// TIA Portal V18 export
// export: Created 2025-12-01T17:50:26.9274774Z, ExportSetting None, DisplayName Totally Integrated Automation Portal, DisplayVersion V18 Update 5, DisplayName TIA Portal Openness, DisplayVersion V18 Update 5, DisplayName TIA Portal Teamcenter Gateway, DisplayVersion V18, DisplayName TIA Portal Version Control Interface, DisplayVersion V18, DisplayName STEP 7 Professional, DisplayVersion V18 Update 5, DisplayName STEP 7 Safety, DisplayVersion V18, DisplayName WinCC Professional, DisplayVersion V18 Update 5
FUNCTION_BLOCK "SystemMode"   // FB3000, LAD
TITLE = SystemMode_FB
{ S7_Optimized_Access := 'TRUE' }
AUTHOR : STD
FAMILY : RCS
VERSION : 2.0
// stored: AutoNumber false, MemoryReserve 100, SetENOAutomatically false
   VAR_INPUT
      iPLCRestarted : Bool;
      iEstopAllOK { ExternalAccessible := 'False'; ExternalVisible := 'False'; ExternalWritable := 'False'} : Bool;   // 急停按钮
      iResetFault { ExternalAccessible := 'False'; ExternalVisible := 'False'; ExternalWritable := 'False'} : Bool;   // 故障复位按钮
      iModeSelectType { ExternalAccessible := 'False'; ExternalVisible := 'False'; ExternalWritable := 'False'} : Bool;   // 0=key switch / 1= HMI button
      iManual { ExternalAccessible := 'False'; ExternalVisible := 'False'; ExternalWritable := 'False'} : Bool;   // Key switch signal,1=Manual / Key switch signal,1=Manual Mode
      iAuto { ExternalAccessible := 'False'; ExternalVisible := 'False'; ExternalWritable := 'False'} : Bool;   // Key switch signal,1=Auto / Key switch signal,1=Auto Mode
      iStep { ExternalAccessible := 'False'; ExternalVisible := 'False'; ExternalWritable := 'False'} : Bool;   // Step mode / Auto Step Mode
      iOneCycle : Bool;   // OneCycle / Auto One Cycle Mode
      iHMIModeSelect { ExternalAccessible := 'False'; ExternalVisible := 'False'; ExternalWritable := 'False'} : Int;   // HMI button signal,1=Manual / 2=Auto/3=OneCycle/4=Step / HMI button signal,1=Manual / 2=Auto / 3=Step / 4=OneCyc
      iControlOnMonitor { ExternalAccessible := 'False'; ExternalVisible := 'False'; ExternalWritable := 'False'} : Bool;   // 安全继电器ControlOn监控
      iSafetyDoor { ExternalAccessible := 'False'; ExternalVisible := 'False'; ExternalWritable := 'False'} : Bool;
      iLightCurtain { ExternalAccessible := 'False'; ExternalVisible := 'False'; ExternalWritable := 'False'} : Bool;
      iSafetyByPass : Bool;
      iMainPressureSwitch { ExternalAccessible := 'False'; ExternalVisible := 'False'; ExternalWritable := 'False'} : Bool;   // 主气源开关监控
      iFixtureOK { ExternalAccessible := 'False'; ExternalVisible := 'False'; ExternalWritable := 'False'} : Bool;   // fixture ok
      iChangeOverOK { ExternalAccessible := 'False'; ExternalVisible := 'False'; ExternalWritable := 'False'} : Bool;   // changer over is ok
      iInitializationOK { ExternalAccessible := 'False'; ExternalVisible := 'False'; ExternalWritable := 'False'} : Bool;   // initialization is ok
      iAllDeviceOK { ExternalAccessible := 'False'; ExternalVisible := 'False'; ExternalWritable := 'False'} : Bool;   // all device is ready
      iAlarmOn : Bool;   // 设备故障
      iFlowRun : Bool;   // 设备运行
   END_VAR
   VAR_OUTPUT
      oReset { ExternalAccessible := 'False'; ExternalVisible := 'False'; ExternalWritable := 'False'} : Bool;   // 系统复位信号
      oEStopOK { ExternalAccessible := 'False'; ExternalVisible := 'False'; ExternalWritable := 'False'} : Bool;   // 系统急停控制信号
      oManualMode { ExternalAccessible := 'False'; ExternalVisible := 'False'; ExternalWritable := 'False'} : Bool;   // 手动模式信号
      oAutoMode { ExternalAccessible := 'False'; ExternalVisible := 'False'; ExternalWritable := 'False'} : Bool;   // 自动模式信号
      oOneCycleMode : Bool;   // 单次循环
      oStepMode { ExternalAccessible := 'False'; ExternalVisible := 'False'; ExternalWritable := 'False'} : Bool;
      oRun { ExternalAccessible := 'False'; ExternalVisible := 'False'; ExternalWritable := 'False'} : Bool;   // 系统运行就绪信号 / Control On and all Safety function OK
      "oEnable alarm" : Bool;
      oControlON { ExternalAccessible := 'False'; ExternalVisible := 'False'; ExternalWritable := 'False'} : Bool;   // PowerON
      oMainPressureOK { ExternalAccessible := 'False'; ExternalVisible := 'False'; ExternalWritable := 'False'} : Bool;   // air pressure
      oSafetyDoorOK { ExternalAccessible := 'False'; ExternalVisible := 'False'; ExternalWritable := 'False'} : Bool;   // 安全门关闭
      oLightCurtainOK { ExternalAccessible := 'False'; ExternalVisible := 'False'; ExternalWritable := 'False'} : Bool;   // 光栅
      oReady : Bool;   // 用于流程控制 / In AutoMode and all condition ok, machine can auto running
      oMode { ExternalAccessible := 'False'; ExternalVisible := 'False'; ExternalWritable := 'False'} : Int;   // 0NA,1Manual, 2Auto, 3Step, 4OneCycle, 5Runn, 6Error
      oStatus : Int;   // 0NotReady, 1Ready, 2AutoRunning, 3EStop, 4Alarm
   END_VAR
   VAR
      sRunT { S7_SetPoint := 'True'} : TON_TIME;
      sPressureTOF { S7_SetPoint := 'True'} : TOF_TIME;
      sChangeOverTOF { S7_SetPoint := 'True'} : TOF_TIME;
      sChangeOverOK { S7_SetPoint := 'True'} : Bool;
   END_VAR
   VAR_TEMP
      tAlwaysOn : Bool;
   END_VAR
   VAR_TEMP   // added for the SCL form of the ladder/FBD networks
      _w1 : Bool;
      _w2 : Bool;
      _w3 : Bool;
   END_VAR
BEGIN

REGION Network 1: AlwaysOn
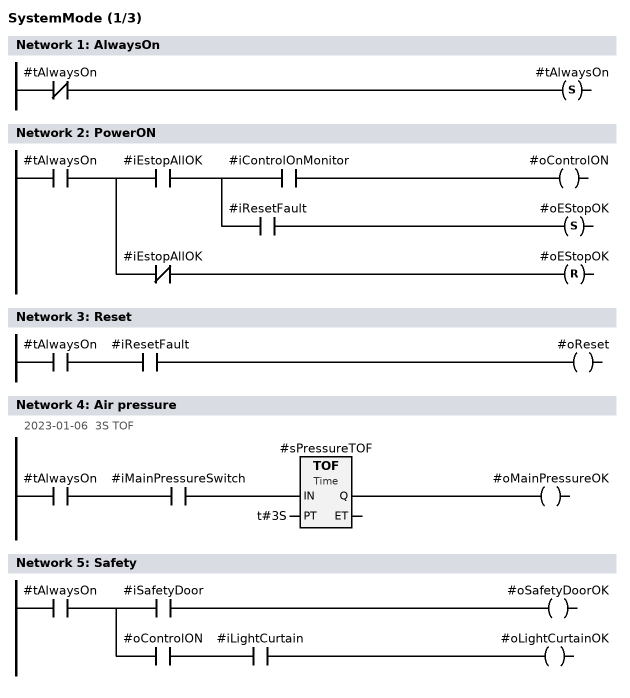
   RUNG wire#powerrail
      I_Contact( #tAlwaysOn )
      S_Coil( #tAlwaysOn )
   END_RUNG
   // the same network as SCL:
   IF NOT #tAlwaysOn THEN #tAlwaysOn := TRUE; END_IF;
END_REGION

REGION Network 2: PowerON
   RUNG wire#powerrail
      Contact( #tAlwaysOn )
      wire#w1
      Contact( #iEstopAllOK )
      wire#w2
      Contact( #iControlOnMonitor )
      Coil( #oControlON )
   END_RUNG
   RUNG wire#w2
      Contact( #iResetFault )
      S_Coil( #oEStopOK )
   END_RUNG
   RUNG wire#w1
      I_Contact( #iEstopAllOK )
      R_Coil( #oEStopOK )
   END_RUNG
   // the same network as SCL:
   #_w1 := #tAlwaysOn AND #iEstopAllOK;
   #oControlON := #_w1 AND #iControlOnMonitor;
   IF #_w1 AND #iResetFault THEN #oEStopOK := TRUE; END_IF;
   IF #tAlwaysOn AND NOT #iEstopAllOK THEN #oEStopOK := FALSE; END_IF;
END_REGION

REGION Network 3: Reset
   RUNG wire#powerrail
      Contact( #tAlwaysOn )
      Contact( #iResetFault )
      Coil( #oReset )
   END_RUNG
   // the same network as SCL:
   #oReset := #tAlwaysOn AND #iResetFault;
END_REGION

REGION Network 4: Air pressure
   // 2023-01-06  3S TOF
   RUNG wire#powerrail
      Contact( #tAlwaysOn )
      Contact( #iMainPressureSwitch )
      { S7_Templates := "time_type := Time" } #sPressureTOF.TOF(pt := t#3S, et =>)
      Coil( #oMainPressureOK )
   END_RUNG
   // the same network as SCL:
   #sPressureTOF(IN := #tAlwaysOn AND #iMainPressureSwitch, PT := t#3S);   // TOF
   #oMainPressureOK := #sPressureTOF.Q;
END_REGION

REGION Network 5: Safety
   RUNG wire#powerrail
      Contact( #tAlwaysOn )
      wire#w1
      Contact( #iSafetyDoor )
      Coil( #oSafetyDoorOK )
   END_RUNG
   RUNG wire#w1
      Contact( #oControlON )
      Contact( #iLightCurtain )
      Coil( #oLightCurtainOK )
   END_RUNG
   // the same network as SCL:
   #oSafetyDoorOK := #tAlwaysOn AND #iSafetyDoor;
   #oLightCurtainOK := #tAlwaysOn AND #oControlON AND #iLightCurtain;
END_REGION

REGION Network 6: Mode
   // 0NA,1Manual, 2Auto, 3Step, 4OneCycle, 5Runn, 6Error
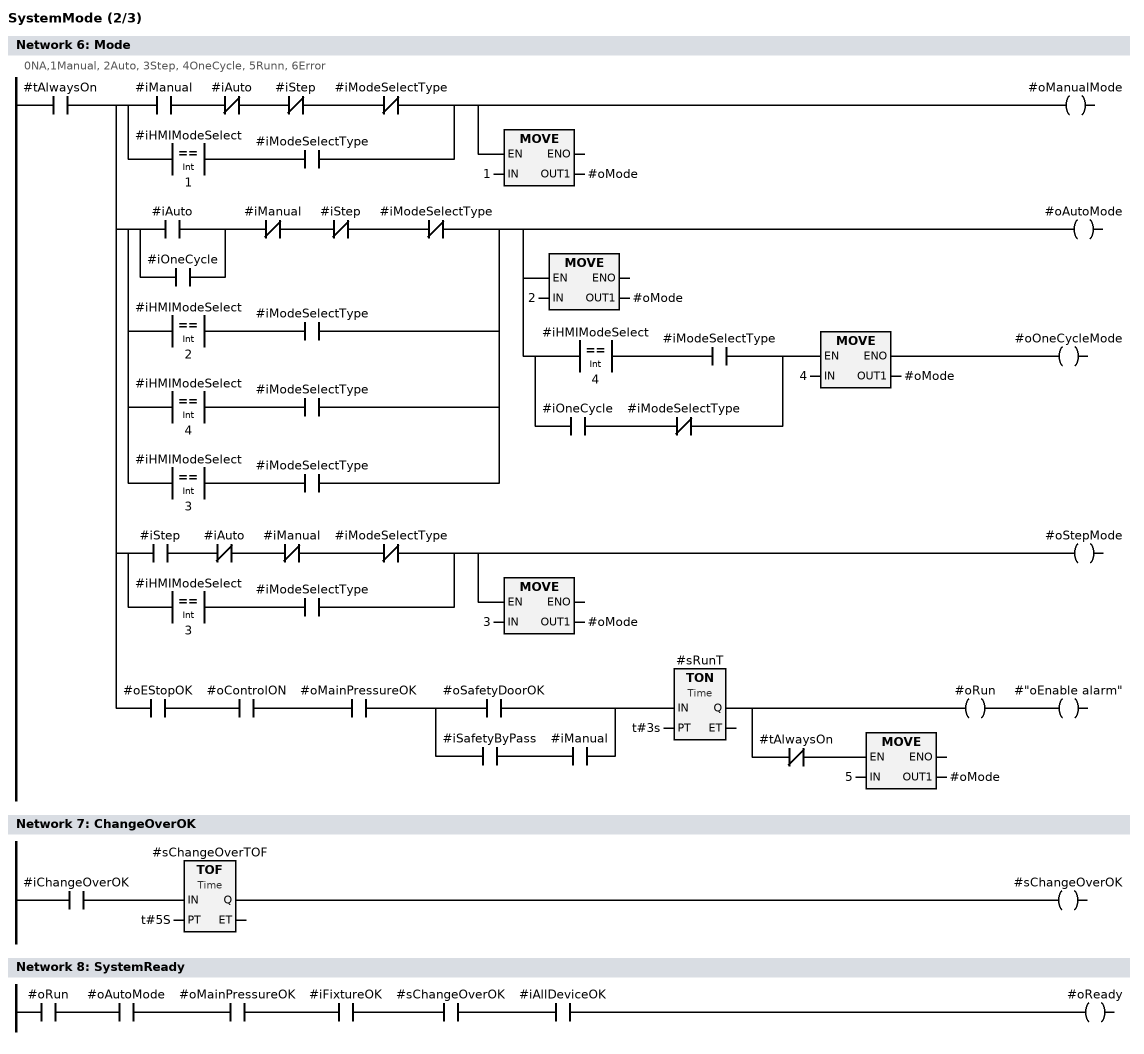
   RUNG wire#powerrail
      Contact( #tAlwaysOn )
      wire#w1
      Contact( #iManual )
      I_Contact( #iAuto )
      I_Contact( #iStep )
      I_Contact( #iModeSelectType )
      wire#w2
      Coil( #oManualMode )
   END_RUNG
   RUNG wire#w1
      { S7_Templates := "SrcType := Int" } EQ_Contact(in1 := #iHMIModeSelect, in2 := 1)
      Contact( #iModeSelectType )
   END_RUNG wire#w2
   RUNG wire#w2
      { S7_GenerateENO := "TRUE" } Move(in := 1, out1 => #oMode)
   END_RUNG
   RUNG wire#w1
      Contact( #iAuto )
      wire#w3
      I_Contact( #iManual )
      I_Contact( #iStep )
      I_Contact( #iModeSelectType )
      wire#w4
      Coil( #oAutoMode )
   END_RUNG
   RUNG wire#w1
      Contact( #iOneCycle )
   END_RUNG wire#w3
   RUNG wire#w1
      { S7_Templates := "SrcType := Int" } EQ_Contact(in1 := #iHMIModeSelect, in2 := 2)
      Contact( #iModeSelectType )
   END_RUNG wire#w4
   RUNG wire#w1
      { S7_Templates := "SrcType := Int" } EQ_Contact(in1 := #iHMIModeSelect, in2 := 4)
      Contact( #iModeSelectType )
   END_RUNG wire#w4
   RUNG wire#w1
      { S7_Templates := "SrcType := Int" } EQ_Contact(in1 := #iHMIModeSelect, in2 := 3)
      Contact( #iModeSelectType )
   END_RUNG wire#w4
   RUNG wire#w4
      { S7_GenerateENO := "TRUE" } Move(in := 2, out1 => #oMode)
   END_RUNG
   RUNG wire#w4
      { S7_Templates := "SrcType := Int" } EQ_Contact(in1 := #iHMIModeSelect, in2 := 4)
      Contact( #iModeSelectType )
      wire#w5
      { S7_GenerateENO := "TRUE" } Move(in := 4, out1 => #oMode)
      Coil( #oOneCycleMode )
   END_RUNG
   RUNG wire#w4
      Contact( #iOneCycle )
      I_Contact( #iModeSelectType )
   END_RUNG wire#w5
   RUNG wire#w1
      Contact( #iStep )
      I_Contact( #iAuto )
      I_Contact( #iManual )
      I_Contact( #iModeSelectType )
      wire#w6
      Coil( #oStepMode )
   END_RUNG
   RUNG wire#w1
      { S7_Templates := "SrcType := Int" } EQ_Contact(in1 := #iHMIModeSelect, in2 := 3)
      Contact( #iModeSelectType )
   END_RUNG wire#w6
   RUNG wire#w6
      { S7_GenerateENO := "TRUE" } Move(in := 3, out1 => #oMode)
   END_RUNG
   RUNG wire#w1
      Contact( #oEStopOK )
      Contact( #oControlON )
      Contact( #oMainPressureOK )
      wire#w7
      Contact( #oSafetyDoorOK )
      wire#w8
      { S7_Templates := "time_type := Time" } #sRunT.TON(pt := t#3s, et =>)
      wire#w9
      Coil( #oRun )
      Coil( #"oEnable alarm" )
   END_RUNG
   RUNG wire#w7
      Contact( #iSafetyByPass )
      Contact( #iManual )
   END_RUNG wire#w8
   RUNG wire#w9
      I_Contact( #tAlwaysOn )
      { S7_GenerateENO := "TRUE" } Move(in := 5, out1 => #oMode)
   END_RUNG
   // the same network as SCL:
   // ENO of a box is taken as its EN; it also drops when the box reports an error
   #oManualMode := #tAlwaysOn AND ((#iManual AND NOT #iAuto AND NOT #iStep AND NOT #iModeSelectType) OR ((#iHMIModeSelect = 1) AND #iModeSelectType));
   IF #oManualMode THEN #oMode := 1; END_IF;
   #oAutoMode := #tAlwaysOn AND (((#iAuto OR #iOneCycle) AND NOT #iManual AND NOT #iStep AND NOT #iModeSelectType) OR ((#iHMIModeSelect = 2) AND #iModeSelectType) OR ((#iHMIModeSelect = 4) AND #iModeSelectType) OR ((#iHMIModeSelect = 3) AND #iModeSelectType));
   IF #oAutoMode THEN #oMode := 2; END_IF;
   #_w1 := #oAutoMode AND (((#iHMIModeSelect = 4) AND #iModeSelectType) OR (#iOneCycle AND NOT #iModeSelectType));
   IF #_w1 THEN #oMode := 4; END_IF;
   #oOneCycleMode := #_w1;
   #oStepMode := #tAlwaysOn AND ((#iStep AND NOT #iAuto AND NOT #iManual AND NOT #iModeSelectType) OR ((#iHMIModeSelect = 3) AND #iModeSelectType));
   IF #oStepMode THEN #oMode := 3; END_IF;
   #sRunT(IN := #tAlwaysOn AND #oEStopOK AND #oControlON AND #oMainPressureOK AND (#oSafetyDoorOK OR (#iSafetyByPass AND #iManual)),   // TON
          PT := t#3s);
   #oRun := #sRunT.Q;
   #"oEnable alarm" := #sRunT.Q;
   IF #sRunT.Q AND NOT #tAlwaysOn THEN #oMode := 5; END_IF;
END_REGION

REGION Network 7: ChangeOverOK
   RUNG wire#powerrail
      Contact( #iChangeOverOK )
      { S7_Templates := "time_type := Time" } #sChangeOverTOF.TOF(pt := t#5S, et =>)
      Coil( #sChangeOverOK )
   END_RUNG
   // the same network as SCL:
   #sChangeOverTOF(IN := #iChangeOverOK, PT := t#5S);   // TOF
   #sChangeOverOK := #sChangeOverTOF.Q;
END_REGION

REGION Network 8: SystemReady
   RUNG wire#powerrail
      Contact( #oRun )
      Contact( #oAutoMode )
      Contact( #oMainPressureOK )
      Contact( #iFixtureOK )
      Contact( #sChangeOverOK )
      Contact( #iAllDeviceOK )
      Coil( #oReady )
   END_RUNG
   // the same network as SCL:
   #oReady := #oRun AND #oAutoMode AND #oMainPressureOK AND #iFixtureOK AND #sChangeOverOK AND #iAllDeviceOK;
END_REGION

REGION Network 9: SystemStatus
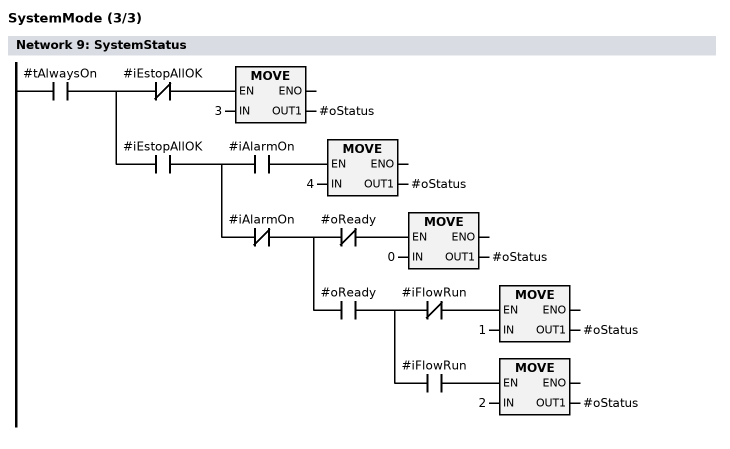
   RUNG wire#powerrail
      Contact( #tAlwaysOn )
      wire#w1
      I_Contact( #iEstopAllOK )
      Move(in := 3, out1 => #oStatus)
   END_RUNG
   RUNG wire#w1
      Contact( #iEstopAllOK )
      wire#w2
      Contact( #iAlarmOn )
      Move(in := 4, out1 => #oStatus)
   END_RUNG
   RUNG wire#w2
      I_Contact( #iAlarmOn )
      wire#w3
      I_Contact( #oReady )
      Move(in := 0, out1 => #oStatus)
   END_RUNG
   RUNG wire#w3
      Contact( #oReady )
      wire#w4
      I_Contact( #iFlowRun )
      Move(in := 1, out1 => #oStatus)
   END_RUNG
   RUNG wire#w4
      Contact( #iFlowRun )
      Move(in := 2, out1 => #oStatus)
   END_RUNG
   // the same network as SCL:
   IF #tAlwaysOn AND NOT #iEstopAllOK THEN #oStatus := 3; END_IF;
   #_w1 := #tAlwaysOn AND #iEstopAllOK;
   IF #_w1 AND #iAlarmOn THEN #oStatus := 4; END_IF;
   #_w2 := #_w1 AND NOT #iAlarmOn;
   IF #_w2 AND NOT #oReady THEN #oStatus := 0; END_IF;
   #_w3 := #_w2 AND #oReady;
   IF #_w3 AND NOT #iFlowRun THEN #oStatus := 1; END_IF;
   IF #_w3 AND #iFlowRun THEN #oStatus := 2; END_IF;
END_REGION
END_FUNCTION_BLOCK
